FUNCTION_BLOCK Test_LTrimEx_HandlesTrimmingManyChars EXTENDS T_UnitTestBase
VAR_INPUT
END_VAR
VAR_OUTPUT
END_VAR
VAR
    SubjectString : T_MaxString := 'Badger';
END_VAR

{attribute 'analysis' := '-33'} // inhibit unused variable warning
METHOD RunTest
IF Retest THEN
	SUPER^.Init();
END_IF

IF TestCompleted THEN
	RETURN;
END_IF

AssertEquals_STRING(Expected := '',
                    Actual   := F_LTrimEx(n := 20, str := SubjectString),
                    Message  := 'F_LTrimEx(SubjectString)');

TestCompleted := TRUE;
END_METHOD

END_FUNCTION_BLOCK

(* stored: Version 1.1.0.1, ProductVersion 3.1.4024.12
   POU Test_LTrimEx_HandlesTrimmingManyChars: Id {08eb4c07-0ad9-078b-191f-cb0e27e2cd67}, SpecialFunc None
   Method RunTest: Id {836a83cb-df96-004f-3211-73789ed47d7b} *)
